FUNCTION_BLOCK sumreal_3 (* Basic FB with empty ECC *)
  (* Standard: 61499-2 *)
  (* Version 1.0, 2021-03-15, Lenovo *)
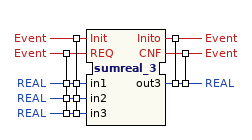
  EVENT_INPUT
    Init WITH in1, in2, in3;
    REQ WITH in1, in2, in3;
  END_EVENT
  EVENT_OUTPUT
    Inito WITH out3;
    CNF WITH out3;
  END_EVENT
  VAR_INPUT
    in1 : REAL;
    in2 : REAL;
    in3 : REAL;
  END_VAR
  VAR_OUTPUT
    out3 : REAL;
  END_VAR
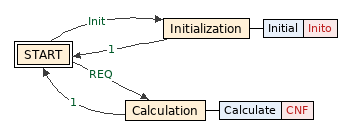
  EC_STATES
    START; (* Initial State *)
    Initialization : Initial -> Inito;
    Calculation : Calculate -> CNF;
  END_STATES
  EC_TRANSITIONS
    START TO Initialization := Init;
    Initialization TO START := 1;
    START TO Calculation := REQ;
    Calculation TO START := 1;
  END_TRANSITIONS
  ALGORITHM Initial IN ST: (* New Algorithm *)

  END_ALGORITHM
  ALGORITHM Calculate IN ST: (* New Algorithm *)
out3:=in1+in2+in3;
  END_ALGORITHM
END_FUNCTION_BLOCK
